(* Logix 5000 project; controller Lab6_Unit18 vendor 1 type 14 code 106 rev 30.11; software revision 30.00 *)

TASK MainTask (continuous, watchdog 500 ms) : MainProgram

MODULES
   Local : vendor 1 type 14 code 106 (Compact 0, rev 30.11)
      I1 : 1769-IQ16 (Compact 1, rev 1.1, Input RPI 20 ms)
      A3 : vendor 1 type 10 code 33 (Compact 3, rev 1.1, Output RPI 80 ms)
      O2 : vendor 1 type 7 code 86 (Compact 2, rev 2.1, Output RPI 20 ms)
END_MODULES

PROGRAM MainProgram   (* main routine MainRoutine *)
VAR
   Black_Mushroomhead_PB : ALIAS FOR Local:1:I.Data.5;
   Blue_Flush_PB : ALIAS FOR Local:1:I.Data.1;
   Blue_Indicator : ALIAS FOR Local:2:O.Data.3;
   Channel3_Input_Data : INT := 180;
   Green_Flush_PB : ALIAS FOR Local:1:I.Data.2;
   Green_Indicator : ALIAS FOR Local:2:O.Data.1;
   Machine_Active : BOOL := 1;
   PVCellPower : REAL := 0.4943848;
   Red_Flush_PB : ALIAS FOR Local:1:I.Data.4;
   Red_Indicator : ALIAS FOR Local:2:O.Data.5;
   Red_Mushroomhead_PB : ALIAS FOR Local:1:I.Data.6;
   Voltage_Input : REAL := 7.03125;
   VoltageSqr : REAL := 49.43848;
   White_Flush_PB : ALIAS FOR Local:1:I.Data.0;
   White_Indicator : ALIAS FOR Local:2:O.Data.4;
   Yellow_Flush_PB : ALIAS FOR Local:1:I.Data.3;
   Yellow_Indicator : ALIAS FOR Local:2:O.Data.2;
END_VAR

ROUTINE MainRoutine   (* ladder *)
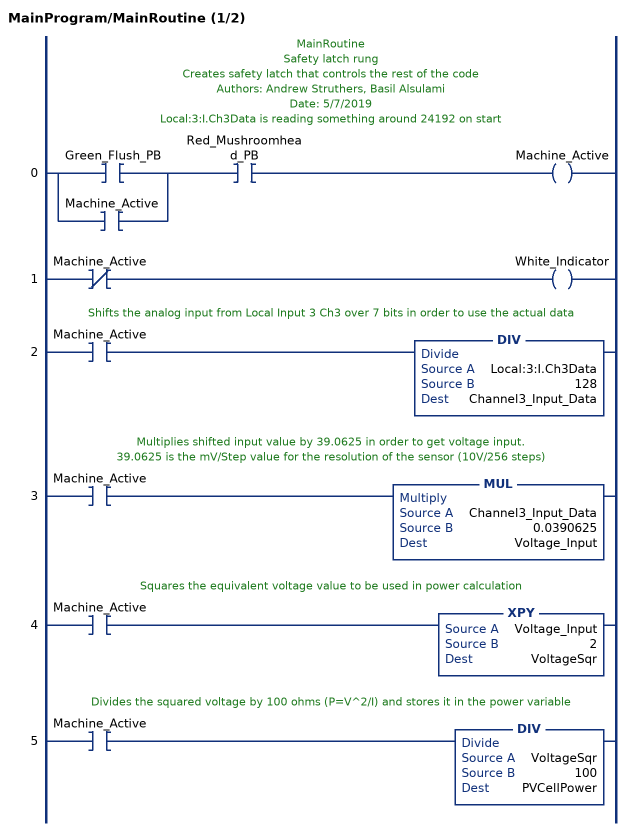
   // MainRoutine
   // Safety latch rung
   // Creates safety latch that controls the rest of the code
   // Authors: Andrew Struthers, Basil Alsulami
   // Date: 5/7/2019
   // Local:3:I.Ch3Data is reading something around 24192 on start
   0: [XIC(Green_Flush_PB) ,XIC(Machine_Active) ]XIC(Red_Mushroomhead_PB)OTE(Machine_Active);
   1: XIO(Machine_Active)OTE(White_Indicator);
   // Shifts the analog input from Local Input 3 Ch3 over 7 bits in order to use the actual data
   2: XIC(Machine_Active)DIV(Local:3:I.Ch3Data,128,Channel3_Input_Data);
   // Multiplies shifted input value by 39.0625 in order to get voltage input.
   // 39.0625 is the mV/Step value for the resolution of the sensor (10V/256 steps)
   3: XIC(Machine_Active)MUL(Channel3_Input_Data,0.0390625,Voltage_Input);
   // Squares the equivalent voltage value to be used in power calculation
   4: XIC(Machine_Active)XPY(Voltage_Input,2,VoltageSqr);
   // Divides the squared voltage by 100 ohms (P=V^2/I) and stores it in the power variable
   5: XIC(Machine_Active)DIV(VoltageSqr,100,PVCellPower);
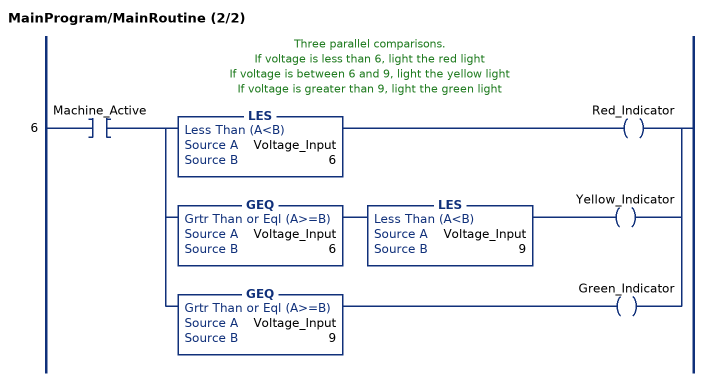
   // Three parallel comparisons.
   // If voltage is less than 6, light the red light
   // If voltage is between 6 and 9, light the yellow light
   // If voltage is greater than 9, light the green light
   6: XIC(Machine_Active)[LES(Voltage_Input,6) OTE(Red_Indicator) ,GEQ(Voltage_Input,6) LES(Voltage_Input,9) OTE(Yellow_Indicator) ,GEQ(Voltage_Input,9) OTE(Green_Indicator) ];
END_ROUTINE
END_PROGRAM
